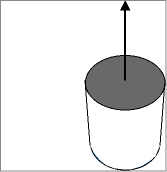
VISUALIZATION VISU_Tube_Top_5  // 167x172
VAR_IN_OUT
	azi : LREAL;
END_VAR
    Ellipse (90,115 70x55)
        p2858320360: azi
    Polygon (85,75) (165,75) (160,145) (157,151) (155,156) (149,161) (141,166) (131,169) (122,169) (114,168) (106,165) (100,160) (94,153) (90,145)
        p2858320360: azi
    Ellipse (85,55 80x55)
        p2858320360: azi
    Polygon (120,10) (125,0) (130,10)
        p2858320360: azi
    Polyline (125,80) (125,10)
        p2858320360: azi
    Polyline (90,145) (85,80)
        p2858320360: azi
    Polyline (160,145) (165,80)
        p2858320360: azi
END_VISUALIZATION

(* stored: Version 1.1.0.1, ProductVersion 3.1.4018.5
   Visu VISU_Tube_Top_5: Id {78e10835-7f7b-4e96-8139-d7c681d7e2c3} *)
